FUNCTION TryConvert_DATE_TO_LWORD : BOOL
VAR_INPUT
	in : DATE;
	out : REFERENCE TO LWORD;
END_VAR

out := DATE_TO_LWORD(in);
TryConvert_DATE_TO_LWORD := TRUE;

END_FUNCTION

(* stored: Version 1.1.0.1, ProductVersion 3.1.4024.12
   POU TryConvert_DATE_TO_LWORD: Id {33dae9f0-2332-45a4-92fc-35278d514ce1}, SpecialFunc None *)
